FUNCTION BufferUdintToReal : REAL
VAR_INPUT
	raw_input :UDINT;
END_VAR
VAR
	temp : DWORD;
END_VAR

temp := UDINT_TO_DWORD(raw_input);
BufferUdintToReal := DWORD_TO_REAL(temp);
temp := BE32_TO_HOST(temp);
MEMCPY(ADR(BufferUdintToReal), ADR(temp), SIZEOF(temp));

END_FUNCTION

(* stored: Version 1.1.0.1, ProductVersion 3.1.4024.9
   POU BufferUdintToReal: Id {460771cb-dcaa-4193-8fd3-80e6a148e719}, SpecialFunc None *)
